{attribute 'hide_all_locals'}
{attribute 'conditionalshow'}
FUNCTION_BLOCK FB_HTTP_Get_Auhofcenter
VAR_INPUT
	{attribute 'hide'}
	bWriteRequest				: BOOL;													//Send a Write Request to the Server
	{attribute 'hide'}
	bReadRequest				: BOOL;													//Send a Read Request to the Server
	{attribute 'hide'}
	arrListOfVariables			: ARRAY[1..100] OF ST_ListOfVariables_Auhofcenter;		//List of Variables what the function must be send or write
	{attribute 'hide'}
	bSend           			: BOOL;													//Send the Request
	{attribute 'hide'}
	tTimeOut					: TIME := T#10S;										//Timer for Timeout
END_VAR
VAR_IN_OUT
	{attribute 'hide'}
    fbClient          			: FB_IotHttpClient;										//HTTP Client Data
END_VAR
VAR_OUTPUT
	{attribute 'hide'}
	bValidResult				: BOOL;													//Valid Result received from Server
	{attribute 'hide'}
    bBusy             			: BOOL;													//Function is Busy
	{attribute 'hide'}
    bError           			: BOOL;													//Error sucess
	{attribute 'hide'}
	byTypeOfLastRequest			: BYTE;													//Type of the last Request. (0 = Read, 1 = Write)
	{attribute 'hide'}
	sContent         			: STRING(7500);											//Received Content
END_VAR
VAR
    fbRequest        		 	: FB_IotHttpRequest;									//Http Function
	RisingEdge        			: R_TRIG;												//Internal positive edge
	timTimeout					: TON;													//Timer for Timeout
   	bGetContentResult 			: BOOL;													//Get Content Result
	byQuantity					: BYTE;													//Quantity of Datapoints
	byLoop						: BYTE;													//Variable foor Loop to prepear the URI
	nState						: UDINT;												//Statemaschine
  	nReqCount					: UDINT;												//Counter requests
    nResCount					: UDINT;												//Counter results
    nValidResCount				: UDINT;												//Counter valid results
    nErrCount					: UDINT;												//Error Counter
	eErrorCode					: ETcIotHttpRequestError;								//Error Code
	sUriStart					: STRING(20);											//Start URI
	sUriComplete				: STRING(2000);											//Complete URI
END_VAR

//Creator : Kai Ebensperger
//Company : Lynus AG
//Date : 15.07.2021
//Version : 1.0.0.0

//With this Function is possible to send a HTTP Get Request to the System in the Auhof Center in Vienna.

//Timer for Timeout
timTimeout(IN:= nState = 1 AND bBusy, PT:= tTimeOut, Q=> , ET=> );
	IF timTimeout.Q THEN nState := 0; bBusy := FALSE; END_IF

RisingEdge(CLK:= bSend);

CASE nState OF
0:
    IF RisingEdge.Q THEN
		
		byQuantity := 0;
			FOR byLoop := 1 TO 100 BY 1 DO
				IF arrListOfVariables[byLoop].sVariableName <> '' THEN byQuantity := byQuantity + 1; END_IF 
			END_FOR
	
		sUriComplete := '';
			//Read Request
			IF bReadRequest THEN 
				sUriStart := '/lynus/read?';
					sUriComplete := sUriStart;
						IF byQuantity <= 100 THEN
							FOR byLoop := 1 TO byQuantity BY 1 DO
								CONCAT2(ADR(sUriComplete),ADR(arrListOfVariables[byLoop].sVariableName),ADR(sUriComplete),SIZEOF(sUriComplete));
									IF byLoop <= (byQuantity - 1) THEN CONCAT2(ADR(sUriComplete),ADR(','),ADR(sUriComplete),SIZEOF(sUriComplete)); END_IF	
							END_FOR
						END_IF
							byTypeOfLastRequest := 0;
			END_IF
				//Write Request
				IF bWriteRequest THEN 
					sUriStart := '/lynus/write?';
						sUriComplete := sUriStart;
							IF byQuantity <= 100 THEN
								FOR byLoop := 1 TO byQuantity BY 1 DO
									CONCAT2(ADR(sUriComplete),ADR(arrListOfVariables[byLoop].sVariableName),ADR(sUriComplete),SIZEOF(sUriComplete));
										CONCAT2(ADR(sUriComplete),ADR('='),ADR(sUriComplete),SIZEOF(sUriComplete));
											IF arrListOfVariables[byLoop].bIsString THEN CONCAT2(ADR(sUriComplete),ADR('"'),ADR(sUriComplete),SIZEOF(sUriComplete)); END_IF 	
												CONCAT2(ADR(sUriComplete),ADR(arrListOfVariables[byLoop].sVariableValue),ADR(sUriComplete),SIZEOF(sUriComplete));
													IF arrListOfVariables[byLoop].bIsString THEN CONCAT2(ADR(sUriComplete),ADR('"'),ADR(sUriComplete),SIZEOF(sUriComplete)); END_IF 			
														IF byLoop <= (byQuantity - 1) THEN CONCAT2(ADR(sUriComplete),ADR(','),ADR(sUriComplete),SIZEOF(sUriComplete)); END_IF	
								END_FOR
							END_IF
								byTypeOfLastRequest := 1;	
				END_IF
		
		bValidResult := FALSE;
		
		IF fbRequest.SendRequest(sUri:= sUriComplete,
								 fbClient:= fbClient, 
									eRequestType:= ETcIotHttpRequestType.HTTP_Get, 0, 0, 0) THEN
			nState:= 1;
			nReqCount:= nReqCount+1;
			bBusy:= TRUE;
			bError:= FALSE;
		END_IF
    END_IF
	
1:
    IF NOT fbRequest.bBusy THEN
       IF NOT fbRequest.bError THEN
            bGetContentResult:= fbRequest.GetContent(pContent:= ADR(sContent), 
                                                     nContentSize:= SIZEOF(sContent), 
                                                     bSetNullTermination:= TRUE);
            IF fbRequest.nStatusCode >= 200 AND fbRequest.nStatusCode < 300 THEN
                	bValidResult := TRUE;
                    nValidResCount:= nValidResCount+1;
                    bError:= FALSE;
               		nResCount:= nResCount+1;
           END_IF
		   		//Error Response from the Server
				IF sContent = 'Error' THEN bError := TRUE; END_IF
        END_IF
			IF fbRequest.bError THEN bError:= TRUE; eErrorCode := fbRequest.eErrorId; END_IF 
			nState:= 0;
			bBusy:= FALSE;
			IF bError THEN
				nErrCount:= nErrCount+1;
			END_IF	
    END_IF
	
END_CASE

END_FUNCTION_BLOCK

(* stored: Version 1.1.0.1, ProductVersion 3.1.4024.9
   POU FB_HTTP_Get_Auhofcenter: Id {99f161aa-48d4-4ea3-9efb-375cd8be7fa0}, SpecialFunc None *)
